// TIA Portal V20 export
// export: Created 2025-12-01T14:56:17.2183909Z, ExportSetting None, DisplayName Totally Integrated Automation Portal, DisplayVersion V20 Update 3, DisplayName TIA Portal Openness, DisplayVersion V20 Update 3, DisplayName TIA Portal Version Control Interface, DisplayVersion V20 Update 3, DisplayName STEP 7 Professional, DisplayVersion V20 Update 3, DisplayName STEP 7 Safety, DisplayVersion V20 Update 2, DisplayName WinCC Basic/Comfort/Advanced, DisplayVersion V20 Update 3, DisplayName WinCC Professional, DisplayVersion V20 Update 3, DisplayName WinCC Unified, DisplayVersion V20 Update 3
TYPE "UDT_Interlock_manual_STV"
   STRUCT
      "byte0.bit0" : Bool;
      "byte0.bit1" : Bool;
      Load_ok : Bool;
      "byte0.bit3" : Bool;
      "byte0.bit4" : Bool;
      "Byte0.bit8" : Bool;
      "Byte0.bit9" : Bool;
      Byte1_bit0 : Bool;
      Byte1_bit1 : Bool;
      Unload_ok : Bool;
      UnloadComplete : Bool;
      Byte1_bit8 : Bool;
      Byte1_bit9 : Bool;
      Byte1_bit10 : Bool;
      Byte1_bit6 : Bool;
      Byte1_bit7 : Bool;
   END_STRUCT;
END_TYPE
